FUNCTION TryConvert_TOD_TO_UDINT : BOOL
VAR_INPUT
	in : TOD;
	out : REFERENCE TO UDINT;
END_VAR

out := TOD_TO_UDINT(in);
TryConvert_TOD_TO_UDINT := TRUE;

END_FUNCTION

(* stored: Version 1.1.0.1, ProductVersion 3.1.4024.12
   POU TryConvert_TOD_TO_UDINT: Id {96c96d5c-e374-4d7f-9e85-ce58a29daea4}, SpecialFunc None *)
